PROGRAM p_ValveSup
VAR
	fbPBT_VGC_01 : FB_VGC;
	fbPBT_VGC_02 : FB_VGC;
	fbPBT_VGC_03 : FB_VGC;
	fbPBT_VGC_04 : FB_VGC;
	
	//vgDownstream: LCLSVACUUMLIB.ST_VG;
END_VAR


vgcPBT_VGC_01.xEXT_OK := TRUE;
fbPBT_VGC_01(iq_stValve:=vgcPBT_VGC_01, i_stDSG:=vgPBT_GCC_04, i_stUSG:=vgPBT_GCC_02, i_xDis_DPIlk:=TRUE);

vgcPBT_VGC_02.xEXT_OK := TRUE;
fbPBT_VGC_02(iq_stValve:=vgcPBT_VGC_02, i_stDSG:=vgPBT_GCC_06, i_stUSG:=vgPBT_GCC_04, i_xDis_DPIlk:=TRUE);

vgcPBT_VGC_03.xEXT_OK := TRUE;
fbPBT_VGC_03(iq_stValve:=vgcPBT_VGC_03, i_stDSG:=vgPBT_GCC_09, i_stUSG:=vgPBT_GCC_07, i_xDis_DPIlk:=TRUE);

vgcPBT_VGC_04.xEXT_OK := TRUE;
//fbPBT_VGC_05(iq_stValve:=vgcPBT_VGC_05, i_stDSG:=vgMON_GCC_04, i_stUSG:=vgPBT_GCC_08, i_xDis_DPIlk:=FALSE);

END_PROGRAM

(* stored: Version 1.1.0.1, ProductVersion 3.1.4020.12
   POU p_ValveSup: Id {a86edaae-e6c6-4d95-8d17-2b811943a0ea}, SpecialFunc None *)
